# EPICS autosave request: apps/chillerApp/Db/anova_settings.req
#
# ANOVA Refrigerated and Heating Circulators - A Series
#
# Author: Wesley Moore
# Date:   July 2014
#

$(P)$(R)PUMPSPD_MENU
$(P)$(R)TEMP_SETPT
$(P)$(R)HIGHLIMIT_SETPT
$(P)$(R)LOWLIMIT_SETPT
